# EPICS autosave request: iocBoot/iocVxWorks/auto_settings_sis.req
file "simple_mca_settings.req",      P=$(P)3820:, M=mca1
file "simple_mca_settings.req",      P=$(P)3820:, M=mca2
file "simple_mca_settings.req",      P=$(P)3820:, M=mca3
file "simple_mca_settings.req",      P=$(P)3820:, M=mca4
file "simple_mca_settings.req",      P=$(P)3820:, M=mca5
file "simple_mca_settings.req",      P=$(P)3820:, M=mca6
file "simple_mca_settings.req",      P=$(P)3820:, M=mca7
file "simple_mca_settings.req",      P=$(P)3820:, M=mca8
file "simple_mca_settings.req",      P=$(P)3820:, M=mca9
file "simple_mca_settings.req",      P=$(P)3820:, M=mca10
file "simple_mca_settings.req",      P=$(P)3820:, M=mca11
file "simple_mca_settings.req",      P=$(P)3820:, M=mca12
file "simple_mca_settings.req",      P=$(P)3820:, M=mca13
file "simple_mca_settings.req",      P=$(P)3820:, M=mca14
file "simple_mca_settings.req",      P=$(P)3820:, M=mca15
file "simple_mca_settings.req",      P=$(P)3820:, M=mca16
file "simple_mca_settings.req",      P=$(P)3820:, M=mca17
file "simple_mca_settings.req",      P=$(P)3820:, M=mca18
file "simple_mca_settings.req",      P=$(P)3820:, M=mca19
file "simple_mca_settings.req",      P=$(P)3820:, M=mca20
file "simple_mca_settings.req",      P=$(P)3820:, M=mca21
file "simple_mca_settings.req",      P=$(P)3820:, M=mca22
file "simple_mca_settings.req",      P=$(P)3820:, M=mca23
file "simple_mca_settings.req",      P=$(P)3820:, M=mca24
file "simple_mca_settings.req",      P=$(P)3820:, M=mca25
file "simple_mca_settings.req",      P=$(P)3820:, M=mca26
file "simple_mca_settings.req",      P=$(P)3820:, M=mca27
file "simple_mca_settings.req",      P=$(P)3820:, M=mca28
file "simple_mca_settings.req",      P=$(P)3820:, M=mca29
file "simple_mca_settings.req",      P=$(P)3820:, M=mca30
file "simple_mca_settings.req",      P=$(P)3820:, M=mca31
file "simple_mca_settings.req",      P=$(P)3820:, M=mca32
file "simple_mca_settings.req",      P=$(P)3801:, M=mca1
file "simple_mca_settings.req",      P=$(P)3801:, M=mca2
file "simple_mca_settings.req",      P=$(P)3801:, M=mca3
file "simple_mca_settings.req",      P=$(P)3801:, M=mca4
file "simple_mca_settings.req",      P=$(P)3801:, M=mca5
file "simple_mca_settings.req",      P=$(P)3801:, M=mca6
file "simple_mca_settings.req",      P=$(P)3801:, M=mca7
file "simple_mca_settings.req",      P=$(P)3801:, M=mca8
file "simple_mca_settings.req",      P=$(P)3801:, M=mca9
file "simple_mca_settings.req",      P=$(P)3801:, M=mca10
file "simple_mca_settings.req",      P=$(P)3801:, M=mca11
file "simple_mca_settings.req",      P=$(P)3801:, M=mca12
file "simple_mca_settings.req",      P=$(P)3801:, M=mca13
file "simple_mca_settings.req",      P=$(P)3801:, M=mca14
file "simple_mca_settings.req",      P=$(P)3801:, M=mca15
file "simple_mca_settings.req",      P=$(P)3801:, M=mca16
file "simple_mca_settings.req",      P=$(P)3801:, M=mca17
file "simple_mca_settings.req",      P=$(P)3801:, M=mca18
file "simple_mca_settings.req",      P=$(P)3801:, M=mca19
file "simple_mca_settings.req",      P=$(P)3801:, M=mca20
file "simple_mca_settings.req",      P=$(P)3801:, M=mca21
file "simple_mca_settings.req",      P=$(P)3801:, M=mca22
file "simple_mca_settings.req",      P=$(P)3801:, M=mca23
file "simple_mca_settings.req",      P=$(P)3801:, M=mca24
file "simple_mca_settings.req",      P=$(P)3801:, M=mca25
file "simple_mca_settings.req",      P=$(P)3801:, M=mca26
file "simple_mca_settings.req",      P=$(P)3801:, M=mca27
file "simple_mca_settings.req",      P=$(P)3801:, M=mca28
file "simple_mca_settings.req",      P=$(P)3801:, M=mca29
file "simple_mca_settings.req",      P=$(P)3801:, M=mca30
file "simple_mca_settings.req",      P=$(P)3801:, M=mca31
file "simple_mca_settings.req",      P=$(P)3801:, M=mca32
